(* CODESYS project module_without_io_mapping.ecp

Project tree, tasks and I/O mapping:
  PFC200_G2_2ETH_RS : 750-8212 PFC200 2ETH RS, WAGO, order no. 0750-8212, version 5.11.1.24
    application Application
      libraries: 
      task PLC_Task (cyclic, interval t#50ms, priority 15) calls PLC_PRG
      program PLC_PRG [ST]
    DeviceAdapter
    Kbus : Kbus, WAGO, version 1.4.0.2
        unmapped channels: K-BUS diagnostics
      _1RO_230_VAC_16A_Pot_free_Relay1NO : 0750-0523, WAGO, order no. 0750-0523, version 0.0.0.11
          unmapped channels: _IN, _OUT
        DeviceAdapter
    MODBUS
      MODBUS : MODBUS, WAGO, order no. n/a, version 1.1.1.15
    Serial
      COM1 : COM1, WAGO, version 0.0.0.19
*)

// PFC200_G2_2ETH_RS/Application/PLC_PRG
PROGRAM PLC_PRG
VAR
END_VAR

END_PROGRAM
